// TIA Portal V16 export
// export: Created 2021-09-08T12:46:07.7571242Z, ExportSetting WithDefaults, DisplayName Totally Integrated Automation Portal, DisplayVersion V16 Update 3, DisplayName TIA Portal Version Control Interface, DisplayVersion V16 Update 2, DisplayName TIA Portal Openness, DisplayVersion V16 Update 3, DisplayName TIA Portal Teamcenter Gateway, DisplayVersion V16, DisplayName STEP 7 Professional, DisplayVersion V16 Update 3, DisplayName STEP 7 Safety, DisplayVersion V16, DisplayName WinCC Advanced, DisplayVersion V16 Update 3
FUNCTION "bitToWord" : Void   // FC5, LAD
{ S7_Optimized_Access := 'TRUE' }
VERSION : 0.1
// stored: AutoNumber true, IsIECCheckEnabled false, SetENOAutomatically false, UDAEnableTagReadback false
   VAR_INPUT
      inBit0 : Bool;
      inBit1 : Bool;
      inBit2 : Bool;
      inBit3 : Bool;
      inBit4 : Bool;
      inBit5 : Bool;
      inBit6 : Bool;
      inBit7 : Bool;
      inBit8 : Bool;
      inBit9 : Bool;
      inBit10 : Bool;
      inBit11 : Bool;
      inBit12 : Bool;
      inBit13 : Bool;
      inBit14 : Bool;
      inBit15 : Bool;
   END_VAR
   VAR_OUTPUT
      outWord : Word;
   END_VAR
BEGIN

REGION Network 1
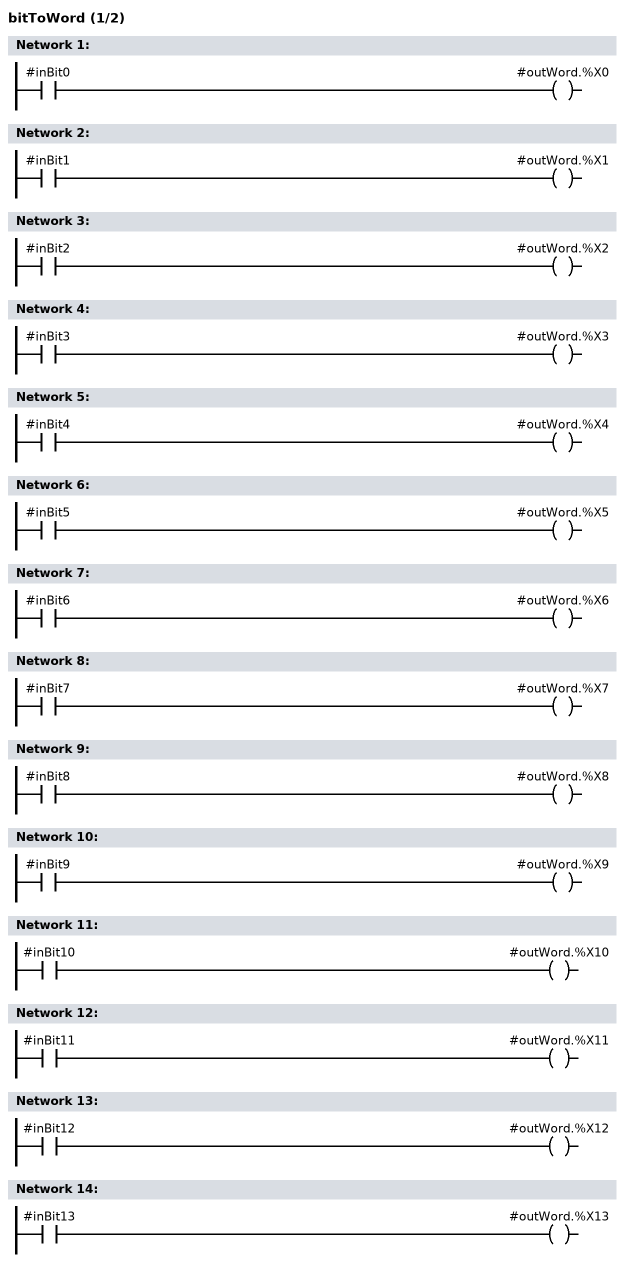
   RUNG wire#powerrail
      Contact( #inBit0 )
      Coil( #outWord.%X0 )
   END_RUNG
   // the same network as SCL:
   #outWord.%X0 := #inBit0;
END_REGION

REGION Network 2
   RUNG wire#powerrail
      Contact( #inBit1 )
      Coil( #outWord.%X1 )
   END_RUNG
   // the same network as SCL:
   #outWord.%X1 := #inBit1;
END_REGION

REGION Network 3
   RUNG wire#powerrail
      Contact( #inBit2 )
      Coil( #outWord.%X2 )
   END_RUNG
   // the same network as SCL:
   #outWord.%X2 := #inBit2;
END_REGION

REGION Network 4
   RUNG wire#powerrail
      Contact( #inBit3 )
      Coil( #outWord.%X3 )
   END_RUNG
   // the same network as SCL:
   #outWord.%X3 := #inBit3;
END_REGION

REGION Network 5
   RUNG wire#powerrail
      Contact( #inBit4 )
      Coil( #outWord.%X4 )
   END_RUNG
   // the same network as SCL:
   #outWord.%X4 := #inBit4;
END_REGION

REGION Network 6
   RUNG wire#powerrail
      Contact( #inBit5 )
      Coil( #outWord.%X5 )
   END_RUNG
   // the same network as SCL:
   #outWord.%X5 := #inBit5;
END_REGION

REGION Network 7
   RUNG wire#powerrail
      Contact( #inBit6 )
      Coil( #outWord.%X6 )
   END_RUNG
   // the same network as SCL:
   #outWord.%X6 := #inBit6;
END_REGION

REGION Network 8
   RUNG wire#powerrail
      Contact( #inBit7 )
      Coil( #outWord.%X7 )
   END_RUNG
   // the same network as SCL:
   #outWord.%X7 := #inBit7;
END_REGION

REGION Network 9
   RUNG wire#powerrail
      Contact( #inBit8 )
      Coil( #outWord.%X8 )
   END_RUNG
   // the same network as SCL:
   #outWord.%X8 := #inBit8;
END_REGION

REGION Network 10
   RUNG wire#powerrail
      Contact( #inBit9 )
      Coil( #outWord.%X9 )
   END_RUNG
   // the same network as SCL:
   #outWord.%X9 := #inBit9;
END_REGION

REGION Network 11
   RUNG wire#powerrail
      Contact( #inBit10 )
      Coil( #outWord.%X10 )
   END_RUNG
   // the same network as SCL:
   #outWord.%X10 := #inBit10;
END_REGION

REGION Network 12
   RUNG wire#powerrail
      Contact( #inBit11 )
      Coil( #outWord.%X11 )
   END_RUNG
   // the same network as SCL:
   #outWord.%X11 := #inBit11;
END_REGION

REGION Network 13
   RUNG wire#powerrail
      Contact( #inBit12 )
      Coil( #outWord.%X12 )
   END_RUNG
   // the same network as SCL:
   #outWord.%X12 := #inBit12;
END_REGION

REGION Network 14
   RUNG wire#powerrail
      Contact( #inBit13 )
      Coil( #outWord.%X13 )
   END_RUNG
   // the same network as SCL:
   #outWord.%X13 := #inBit13;
END_REGION

REGION Network 15
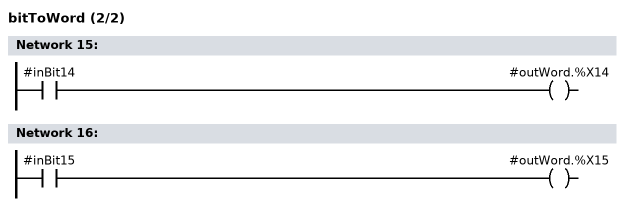
   RUNG wire#powerrail
      Contact( #inBit14 )
      Coil( #outWord.%X14 )
   END_RUNG
   // the same network as SCL:
   #outWord.%X14 := #inBit14;
END_REGION

REGION Network 16
   RUNG wire#powerrail
      Contact( #inBit15 )
      Coil( #outWord.%X15 )
   END_RUNG
   // the same network as SCL:
   #outWord.%X15 := #inBit15;
END_REGION
END_FUNCTION
